TYPE Order_TYP :
STRUCT
	order_num : INT;
	red : INT;
	orange : INT;
	pink : INT;
END_STRUCT
END_TYPE

(* stored: Version 1.1.0.1, ProductVersion 3.1.4024.12
   DUT Order_TYP: Id {faaab30b-846c-09e9-0e01-8e587fd08171} *)
